// TIA Portal V17 export
// export: Created 2026-05-13T14:55:42.260679Z, ExportSetting WithDefaults, DisplayName Totally Integrated Automation Portal, DisplayVersion V17 Update 4, DisplayName TIA Portal Openness, DisplayVersion V17 Update 4, DisplayName TIA Portal Version Control Interface, DisplayVersion V17, DisplayName SINAMICS Startdrive Advanced, DisplayVersion V17, DisplayName SINAMICS Startdrive G130, G150, S120, S150, SINAMICS MV, S210, DisplayVersion V17, DisplayName SINAMICS Startdrive G110M, G120, G120C, G120D, G120P, G115D, DisplayVersion V17, DisplayName STEP 7 Professional, DisplayVersion V17 Update 4, DisplayName STEP 7 Safety, DisplayVersion V17, DisplayName WinCC Professional, DisplayVersion V17 Update 4
ORGANIZATION_BLOCK "Startup"   // OB100, SCL, Startup
TITLE = "Complete Restart"
{ S7_Optimized_Access := 'TRUE' }
VERSION : 0.1
// stored: AutoNumber true, IsIECCheckEnabled false, SetENOAutomatically false
   VAR_INPUT
      LostRetentive : Bool;   // True if retentive data are lost
      LostRTC : Bool;   // True if date and time are lost
   END_VAR
BEGIN
   // === 阀门01 配置 ===
   "DB_Components".Valve01.SwitchCnt := 2;
   "DB_Components".Valve01.RealCnt := 0;
   "DB_Components".Valve01.InfoCnt := 2;
   "DB_Components".Valve01.InfoTitle := '阀门01';
   "DB_Components".Valve01.InfoMessage := '是否确认开启阀门01？';

   // === 电加热01 配置 ===
   "DB_Components".Heater01.SwitchCnt := 1;
   "DB_Components".Heater01.RealCnt := 3;
   "DB_Components".Heater01.InfoCnt := 2;
   "DB_Components".Heater01.InfoTitle := '电加热01';
   "DB_Components".Heater01.InfoMessage := '是否确认开启电加热01？';

   // === 循环风机01 配置 ===
   "DB_Components".Fan01.SwitchCnt := 1;
   "DB_Components".Fan01.RealCnt := 2;
   "DB_Components".Fan01.InfoCnt := 2;
   "DB_Components".Fan01.InfoTitle := '循环风机01';
   "DB_Components".Fan01.InfoMessage := '是否确认开启循环风机01？';
END_ORGANIZATION_BLOCK
